{attribute 'qualified_only'}
{attribute 'strict'}
TYPE E_Xelectrix_Error :
(
	eNoError := 0,
	eModbusTCPError := 1,
	eXelectrixError := 2
);
END_TYPE

(* stored: Version 1.1.0.1, ProductVersion 3.1.4024.9
   DUT E_Xelectrix_Error: Id {bee193e0-ad34-40c7-8bdb-f4d3a0103cb8} *)
